SUBAPPLICATION MSS_Auswahl (* Waehlt per Button die vom Traktor gemeldete Machine Selected Speed (MSS) als Quelle aus, merkt sich die Auswahl persistent im NVS, setzt bei Auswahl die anderen Quellen zurueck und liefert die MSS-Sensordaten nach aussen *)
  (* Standard: 61499-2 *)
  (* Version 1.0, 2026-08-27, Franz *)
  PACKAGE FBs::Baumsetzer::func::Automatik;
  IMPORT NVS_Keys::Key_MSS_Store;
  IMPORT isobus::UT::io::Button::ButtonActivationCode::BT_RELEASED_UNLATCHED;
  IMPORT test::FBs::Baumsetzer::Constants::DefaultPool::Button_MSS;
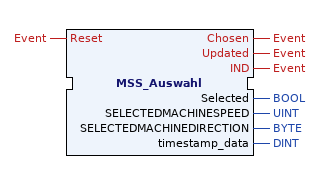
  EVENT_INPUT
    Reset; (* Anforderung von einer der anderen Quellen: eigene Auswahl zuruecksetzen *)
  END_EVENT
  EVENT_OUTPUT
    Chosen; (* Button_MSS wurde gedrueckt: eigene Auswahl setzen und alle anderen Quellen zuruecksetzen *)
    Updated; (* Ausgewaehlt-Status verfuegbar bzw. geaendert (Init-Lesen oder Aenderung); Trigger fuer nachgelagerte Verarbeitung (u.a. Hintergrundfarbe) *)
    IND; (* Neue MSS-Daten empfangen (Indication von I_MSS) *)
  END_EVENT
  VAR_OUTPUT
    Selected : BOOL; (* TRUE wenn MSS aktuell als Geschwindigkeitsquelle ausgewaehlt ist *)
    SELECTEDMACHINESPEED : UINT; (* Vom Traktor gemeldete Machine Selected Speed (PGN 61474, SPN 4305) *)
    SELECTEDMACHINEDIRECTION : BYTE; (* Fahrtrichtung der Machine Selected Speed (PGN 61474, SPN 4309) *)
    timestamp_data : DINT; (* Zeitstempel der letzten MSS-Botschaft *)
  END_VAR
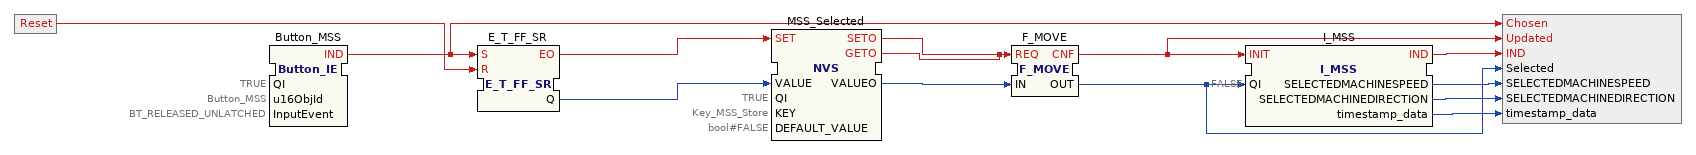
  FBS
    Button_MSS : isobus::UT::io::Button::Button_IE(QI := TRUE, u16ObjId := Button_MSS, InputEvent := BT_RELEASED_UNLATCHED);
    E_T_FF_SR : iec61499::events::E_T_FF_SR;
    MSS_Selected : logiBUS::storage::esp32_nvs::NVS(QI := TRUE, KEY := Key_MSS_Store, DEFAULT_VALUE := bool#FALSE);
    F_MOVE : iec61131::selection::F_MOVE; {SET_ATTRIBUTE(DataType, BOOL)}
    I_MSS : isobus::tecu::I_MSS(QI := FALSE);
  END_FBS
  EVENT_CONNECTIONS
    Button_MSS.IND TO E_T_FF_SR.S;
    Button_MSS.IND TO Chosen;
    Reset TO E_T_FF_SR.R;
    E_T_FF_SR.EO TO MSS_Selected.SET;
    MSS_Selected.SETO TO F_MOVE.REQ;
    MSS_Selected.GETO TO F_MOVE.REQ;
    F_MOVE.CNF TO Updated;
    I_MSS.IND TO IND;
    F_MOVE.CNF TO I_MSS.INIT;
  END_CONNECTIONS
  DATA_CONNECTIONS
    E_T_FF_SR.Q TO MSS_Selected.VALUE;
    MSS_Selected.VALUEO TO F_MOVE.IN;
    F_MOVE.OUT TO I_MSS.QI;
    F_MOVE.OUT TO Selected;
    I_MSS.SELECTEDMACHINESPEED TO SELECTEDMACHINESPEED;
    I_MSS.SELECTEDMACHINEDIRECTION TO SELECTEDMACHINEDIRECTION;
    I_MSS.timestamp_data TO timestamp_data;
  END_CONNECTIONS
END_SUBAPPLICATION
